TYPE MotionParameters_typ :
    STRUCT

        Jerk         : LREAL;                           // mm/s3
        Acceleration : LREAL;                           // mm/s2
        Deceleration : LREAL;                           // mm/s2
        Velocity     : LREAL;                           // mm/s
        Direction    : Tc3_Mc3Definitions.MC_Direction; // MC_Direction
		Gap			 : LREAL;							// mm
		GapMode		 : MC_GAP_CONTROL_MODE := MC_GAP_CONTROL_MODE.mcGapControlModeGroupDefault; // default to mode defined in collision avoidance object

    END_STRUCT
END_TYPE

(* stored: Version 1.1.0.1, ProductVersion 3.1.4026.8
   DUT MotionParameters_typ: Id {bd3dfc46-8034-4584-b9a8-07f88efb1905} *)
